Omron CX-Programmer project NewProject (CX-Programmer 9.61)

# PLC SemifinalPLC: CJ2M CPU11
I/O table (CPU CJ2M-CPU11): rack 0 slot 0 CJ1W-ID211; rack 0 slot 1 CJ1W-OD211

## Global symbols (name address type ; comment)
0.08 BOOL  ; PB Jus Apel
0.00 BOOL  ; PB Start
0.01 BOOL  ; PB Stop
0.07 BOOL  ; PB Jus Jeruk
0.09 BOOL  ; PB Jus Mangga
1.00 BOOL  ; Mixer T1
1.01 BOOL  ; Valve T1
1.02 BOOL  ; Valve T2
1.03 BOOL  ; valve T3
1.04 BOOL  ; Valve T4
1.05 BOOL  ; Pump
1.06 BOOL  ; Heater
1.07 BOOL  ; Solenoid
1.08 BOOL  ; Lampu Merah
1.09 BOOL  ; Lampu Hijau
20.00 BOOL  ; M Jeruk
20.01 BOOL  ; M Apel
20.02 BOOL  ; M Mangga
20.03 BOOL  ; MB Jeruk
20.04 BOOL  ; MB Apel
20.05 BOOL  ; MB Mangga
20.06 BOOL  ; Solenoid State
20.07 BOOL  ; Solenoid State 2
20.08 BOOL  ; State Sensor Berat
20.09 BOOL  ; Lock Off T2
20.10 BOOL  ; Lock OFF T3
20.11 BOOL  ; State TM
20.12 BOOL  ; memory Mixer
D100 CHANNEL  ; Data Barcode
D101 CHANNEL  ; Data Sensor Berat T1
D102 CHANNEL  ; Data Sensor Suhu
D103 CHANNEL  ; Data Sensor Berat TM
T0000 BOOL  ; Timer T2
T0001 BOOL  ; Timer T3
T0002 BOOL  ; Timer Mixer T1
Indikator LampuIndikator
Lampu_Indikator LampuIndikator
PB_Buah LampuIndikator
PB_Buah_ PBBuah
Push_Button_Buah PBBuah
Sensor_Barcode SensorBuah
Sensor_Berat_TM LampuIndikator
Sensor_Berat_TM_ SensorBeratTM
Sensor_State SensorBeratState
Sensor_beratTM SensorBeratTM
Sistem_Heater SistemHeater
Timbangan_Berat_T1 TimbanganT1

## Program Mesin_Jus (cyclic task 0)

### Section Main_Program

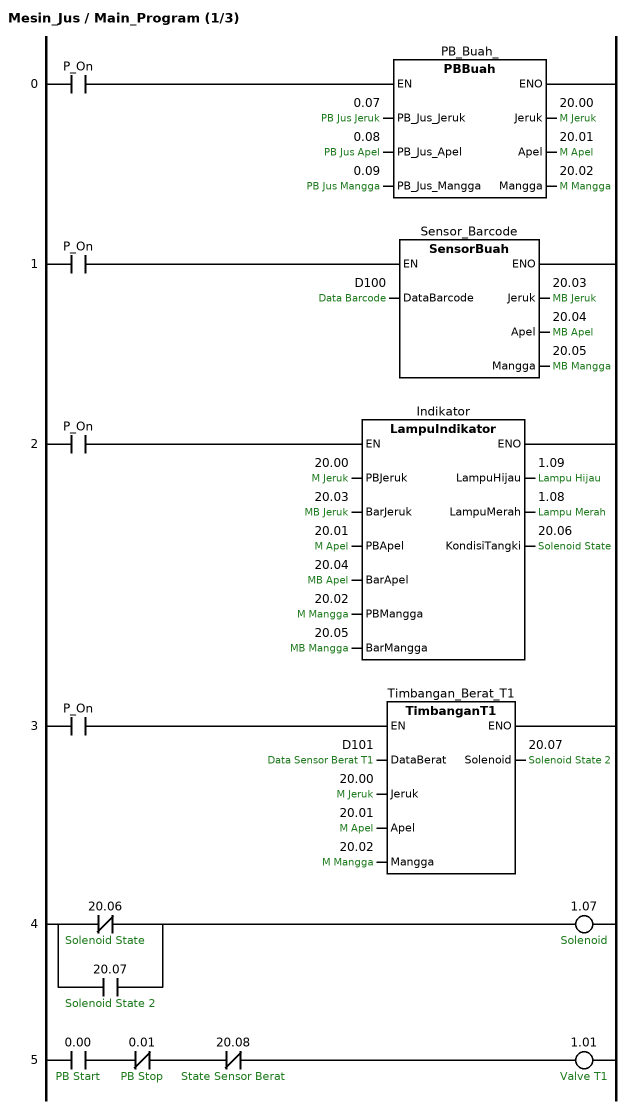
; rung 0
LD P_On
CALL PB_Buah_ : PBBuah (PB_Jus_Jeruk := 0.07, PB_Jus_Apel := 0.08, PB_Jus_Mangga := 0.09, Jeruk => 20.00, Apel => 20.01, Mangga => 20.02)  ; PB Jus Jeruk, PB Jus Apel, PB Jus Mangga, M Jeruk, M Apel, M Mangga
; rung 1
LD P_On
CALL Sensor_Barcode : SensorBuah (DataBarcode := D100, Jeruk => 20.03, Apel => 20.04, Mangga => 20.05)  ; Data Barcode, MB Jeruk, MB Apel, MB Mangga
; rung 2
LD P_On
CALL Indikator : LampuIndikator (PBJeruk := 20.00, BarJeruk := 20.03, PBApel := 20.01, BarApel := 20.04, PBMangga := 20.02, BarMangga := 20.05, LampuHijau => 1.09, LampuMerah => 1.08, KondisiTangki => 20.06)  ; M Jeruk, MB Jeruk, M Apel, MB Apel, M Mangga, MB Mangga, Lampu Hijau, Lampu Merah, Solenoid State
; rung 3
LD P_On
CALL Timbangan_Berat_T1 : TimbanganT1 (DataBerat := D101, Jeruk := 20.00, Apel := 20.01, Mangga := 20.02, Solenoid => 20.07)  ; Data Sensor Berat T1, M Jeruk, M Apel, M Mangga, Solenoid State 2
; rung 4
LDNOT 20.06  ; Solenoid State
OR 20.07  ; Solenoid State 2
OUT 1.07  ; Solenoid
; rung 5
LD 0.00  ; PB Start
ANDNOT 0.01  ; PB Stop
ANDNOT 20.08  ; State Sensor Berat
OUT 1.01  ; Valve T1

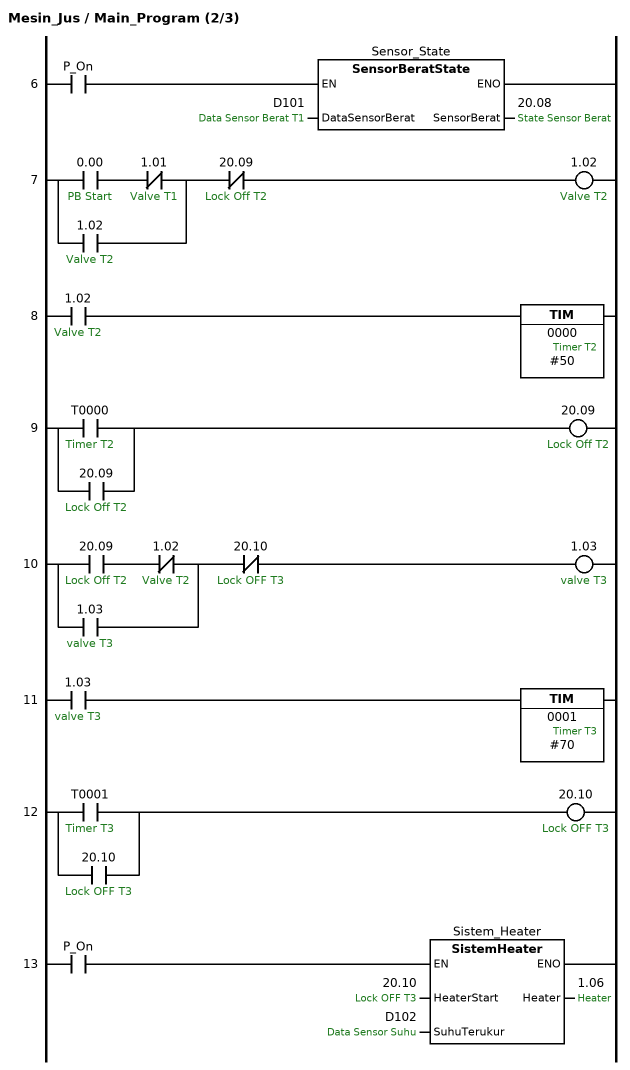
; rung 6
LD P_On
CALL Sensor_State : SensorBeratState (DataSensorBerat := D101, SensorBerat => 20.08)  ; Data Sensor Berat T1, State Sensor Berat
; rung 7
LD 0.00  ; PB Start
ANDNOT 1.01  ; Valve T1
OR 1.02  ; Valve T2
ANDNOT 20.09  ; Lock Off T2
OUT 1.02  ; Valve T2
; rung 8
LD 1.02  ; Valve T2
TIM 0000 #50  ; Timer T2
; rung 9
LD T0000  ; Timer T2
OR 20.09  ; Lock Off T2
OUT 20.09  ; Lock Off T2
; rung 10
LD 20.09  ; Lock Off T2
ANDNOT 1.02  ; Valve T2
OR 1.03  ; valve T3
ANDNOT 20.10  ; Lock OFF T3
OUT 1.03  ; valve T3
; rung 11
LD 1.03  ; valve T3
TIM 0001 #70  ; Timer T3
; rung 12
LD T0001  ; Timer T3
OR 20.10  ; Lock OFF T3
OUT 20.10  ; Lock OFF T3
; rung 13
LD P_On
CALL Sistem_Heater : SistemHeater (HeaterStart := 20.10, SuhuTerukur := D102, Heater => 1.06)  ; Lock OFF T3, Data Sensor Suhu, Heater

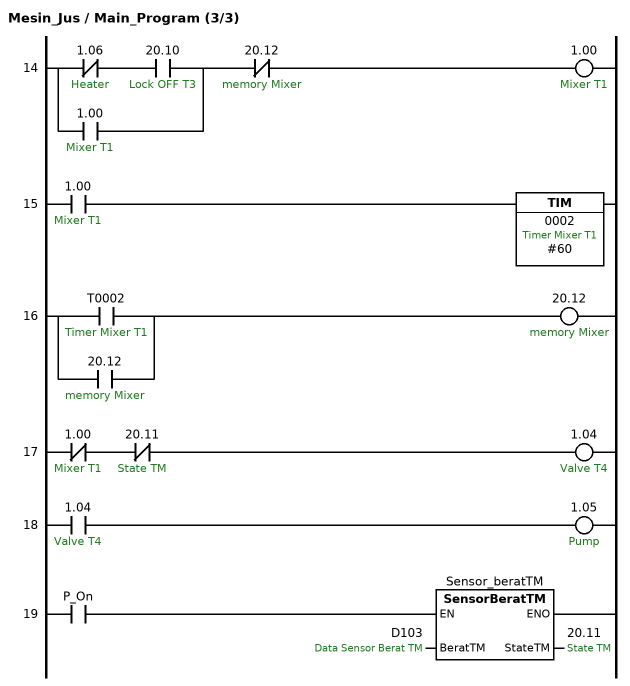
; rung 14
LDNOT 1.06  ; Heater
AND 20.10  ; Lock OFF T3
OR 1.00  ; Mixer T1
ANDNOT 20.12  ; memory Mixer
OUT 1.00  ; Mixer T1
; rung 15
LD 1.00  ; Mixer T1
TIM 0002 #60  ; Timer Mixer T1
; rung 16
LD T0002  ; Timer Mixer T1
OR 20.12  ; memory Mixer
OUT 20.12  ; memory Mixer
; rung 17
LDNOT 1.00  ; Mixer T1
ANDNOT 20.11  ; State TM
OUT 1.04  ; Valve T4
; rung 18
LD 1.04  ; Valve T4
OUT 1.05  ; Pump
; rung 19
LD P_On
CALL Sensor_beratTM : SensorBeratTM (BeratTM := D103, StateTM => 20.11)  ; Data Sensor Berat TM, State TM

### Section END
; rung 0
END(001)

## Function block LampuIndikator
VAR_INPUT
  PBJeruk : BOOL;
  BarJeruk : BOOL;
  PBApel : BOOL;
  BarApel : BOOL;
  PBMangga : BOOL;
  BarMangga : BOOL;
END_VAR
VAR_OUTPUT
  LampuHijau : BOOL;
  LampuMerah : BOOL;
  KondisiTangki : BOOL := TRUE;
END_VAR

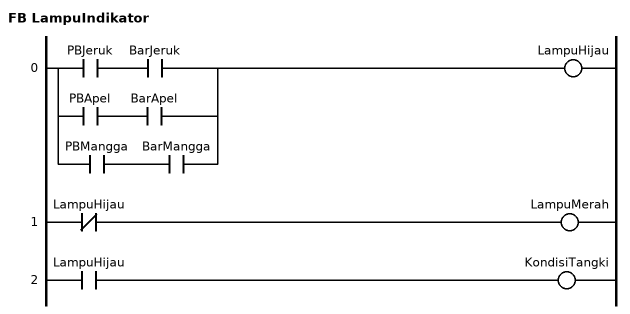
; rung 0
LD PBJeruk
AND BarJeruk
LD PBApel
AND BarApel
ORLD
LD PBMangga
AND BarMangga
ORLD
OUT LampuHijau
; rung 1
LDNOT LampuHijau
OUT LampuMerah
; rung 2
LD LampuHijau
OUT KondisiTangki

## Function block PBBuah
VAR_INPUT
  PB_Jus_Jeruk : BOOL;
  PB_Jus_Apel : BOOL;
  PB_Jus_Mangga : BOOL;
END_VAR
VAR_OUTPUT
  Jeruk : BOOL;
  Apel : BOOL;
  Mangga : BOOL;
END_VAR

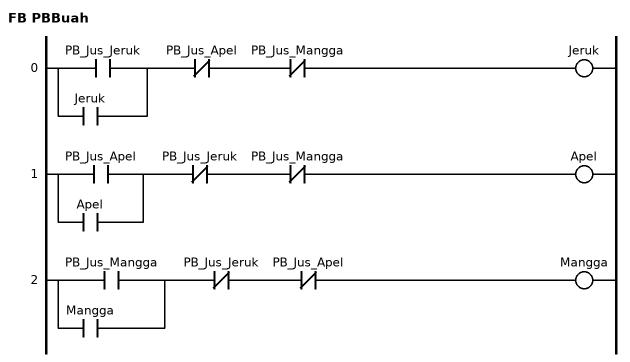
; rung 0
LD PB_Jus_Jeruk
OR Jeruk
ANDNOT PB_Jus_Apel
ANDNOT PB_Jus_Mangga
OUT Jeruk
; rung 1
LD PB_Jus_Apel
OR Apel
ANDNOT PB_Jus_Jeruk
ANDNOT PB_Jus_Mangga
OUT Apel
; rung 2
LD PB_Jus_Mangga
OR Mangga
ANDNOT PB_Jus_Jeruk
ANDNOT PB_Jus_Apel
OUT Mangga

## Function block SensorBeratState
VAR_INPUT
  DataSensorBerat : INT;
END_VAR
VAR_OUTPUT
  SensorBerat : BOOL;
END_VAR
IF DataSensorBerat = 0 THEN
	SensorBerat:= TRUE;
ELSE
	SensorBerat:= FALSE;
END_IF;

## Function block SensorBeratTM
VAR_INPUT
  BeratTM : INT := 6;
END_VAR
VAR_OUTPUT
  StateTM : BOOL;
END_VAR
IF BeratTM=0 THEN
	StateTM:= TRUE;
ELSE
	StateTM:= FALSE;
END_IF;

## Function block SensorBuah
VAR_INPUT
  DataBarcode : INT;
END_VAR
VAR_OUTPUT
  Jeruk : BOOL;
  Apel : BOOL;
  Mangga : BOOL;
END_VAR
IF DataBarcode=678 THEN
	Jeruk:= TRUE;
	Apel:= FALSE;
	Mangga:= FALSE;
ELSIF DataBarcode=768 THEN
	Jeruk:= FALSE;
	Apel:= TRUE;
	Mangga:= FALSE;
ELSIF DataBarcode=876 THEN
	Jeruk:= FALSE;
	Apel:= FALSE;
	Mangga:= TRUE;
ELSE 
	Jeruk:= FALSE;
	Apel:= FALSE;
	Mangga:= FALSE;	
END_IF;

## Function block SistemHeater
VAR_INPUT
  HeaterStart : BOOL;
  SuhuTerukur : INT;
END_VAR
VAR_OUTPUT
  Heater : BOOL;
END_VAR
IF HeaterStart=TRUE AND SuhuTerukur<100 THEN
	Heater:= TRUE;
ELSE
	Heater:= FALSE;
END_IF;

## Function block SistemStarting
VAR_INPUT
  PBStart : BOOL;
  PBStop : BOOL;
END_VAR
VAR_OUTPUT
  No : BOOL;
END_VAR

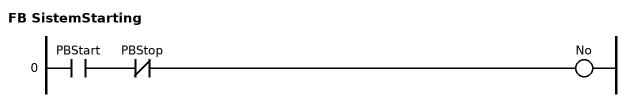
; rung 0
LD PBStart
ANDNOT PBStop
OUT No

## Function block TimbanganT1
VAR_INPUT
  DataBerat : INT;
  Jeruk : BOOL;
  Apel : BOOL;
  Mangga : BOOL;
END_VAR
VAR_OUTPUT
  Solenoid : BOOL;
END_VAR
IF Jeruk=TRUE AND DataBerat=6 THEN
	Solenoid:=TRUE;
ELSIF Apel=TRUE AND DataBerat=9 THEN
	Solenoid:=TRUE;
ELSIF Mangga=TRUE AND DataBerat=12 THEN
	Solenoid:=TRUE;
ELSE
	Solenoid:= FALSE;
END_IF;